// TIA Portal V21 export
FUNCTION "Block_1wadawd" : Void   // FC1, LAD
{ S7_Optimized_Access := 'TRUE' }
// stored: SetENOAutomatically false
BEGIN
END_FUNCTION
